FUNCTION_BLOCK CM_ChkService (* Basic Function Block Type *)
  (* Standard: 61499-2 *)
  (* Version 0.0, 2014-09-04, EQUEROL, UJI *)
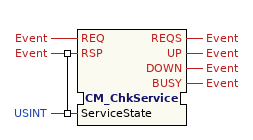
  EVENT_INPUT
    REQ; (* Normal Execution Request *)
    RSP WITH ServiceState; (* Service State response *)
  END_EVENT
  EVENT_OUTPUT
    REQS; (* Request Service State *)
    UP; (* Service is UP *)
    DOWN; (* Service is down *)
    BUSY; (* Service is up but busy *)
  END_EVENT
  VAR_INPUT
    ServiceState : USINT; (* CNC Service State *)
  END_VAR
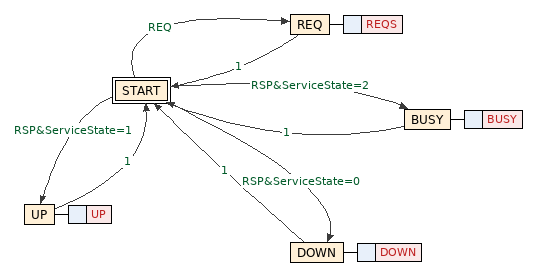
  EC_STATES
    START; (* Initial State *)
    REQ : -> REQS;
    UP : -> UP;
    DOWN : -> DOWN;
    BUSY : -> BUSY;
  END_STATES
  EC_TRANSITIONS
    REQ TO START := 1;
    START TO REQ := REQ;
    START TO UP := RSP&ServiceState=1;
    START TO DOWN := RSP&ServiceState=0;
    START TO BUSY := RSP&ServiceState=2;
    BUSY TO START := 1;
    DOWN TO START := 1;
    UP TO START := 1;
  END_TRANSITIONS
  ALGORITHM INIT IN ST: (* Initialization algorithm *)

  END_ALGORITHM
  ALGORITHM REQ IN ST: (* Normally executed algorithm *)

  END_ALGORITHM
END_FUNCTION_BLOCK
